{attribute 'GeneratedUsingTerminal: EK1122-0000-0018'}
{attribute addProperty BoxType "EK1122-0000-0018"}
{attribute addProperty Id "Beckhoff_EL19xxsub_EK1100EK1100_AB5A94672"}
{attribute addProperty CRC "3302961103"}
{attribute addProperty Size "2"}
TYPE Beckhoff_EL19xxEK1122_C4DF2FCF EXTENDS EK1122_AB5A9467 :
STRUCT
	{attribute addProperty Name "Beckhoff_EL19xxsub_EK1100"}
	Beckhoff_EL19xxsub_EK1100 : EK1100_AB5A9467;
END_STRUCT
END_TYPE

(* stored: Version 1.2.0.0, ProductVersion 3.1.4024.9
   DUT Beckhoff_EL19xxEK1122_C4DF2FCF: Id {c3026943-f97e-406b-87e0-2718988377b3} *)
